{attribute 'reflection'} 
FUNCTION_BLOCK PUBLIC FB_Testsuites EXTENDS FB_Base IMPLEMENTS I_Testsuites
VAR_INPUT
	fbList:				FB_ListTestsuite;
END_VAR
VAR_OUTPUT
END_VAR
VAR
	stTestsuites:    	ST_Testsuites;
	bSave: 				BOOL;
	sFilePathName:		STRING(255):= 'C:\report.xml';

	fbXml:				FB_XmlDomParser;
	testsuites:			PVOID;
END_VAR

SUPER^();


fbXml.SaveDocumentToFile(sFilePathName, bSave);

METHOD PROTECTED M_Started : BOOL
VAR_INPUT
END_VAR

VAR
	nIndex: DINT;
END_VAR
M_Started:= TRUE;
WHILE nIndex < fbList.P_Length DO
	M_Started:= M_Started AND (fbList.M_Get(nIndex).P_State = E_Base.Stopped);
	nIndex:= nIndex + 1;
END_WHILE
END_METHOD

METHOD PROTECTED M_Starting : BOOL
VAR_INPUT
END_VAR

VAR
	nIndex: DINT;
END_VAR
CASE nState OF
	0:
		IF 	SUPER^.M_Starting() THEN
			fbXml.NewDocument();
			stTestsuites.sName:= M_GetName(sInstancePath);
			stTestsuites.nTests:= 0;
			stTestsuites.nFailures:= 0;
			stTestsuites.nErrors:= 0;
			stTestsuites.nSkipped:= 0;
			stTestsuites.nAssertions:= 0;
			stTestsuites.fTime:= 0.0;
			nState:= 1;
		END_IF
		
	1:
		testsuites:= fbXml.AppendNode(fbXml.GetDocumentNode(), 'testsuites');
		fbXml.AppendAttribute(testsuites, 'name', stTestsuites.sName);					// name        Name of the entire test run  
		fbXml.AppendAttributeAsInt(testsuites, 'tests', stTestsuites.nTests);			// tests       Total number of tests in this file    
		fbXml.AppendAttributeAsInt(testsuites, 'failures', stTestsuites.nFailures);		// failures    Total number of failed tests in this file 
		fbXml.AppendAttributeAsInt(testsuites, 'errors', stTestsuites.nErrors);			// errors      Total number of errored tests in this file     
		fbXml.AppendAttributeAsInt(testsuites, 'skipped', stTestsuites.nSkipped);		// skipped     Total number of skipped tests in this file    
		fbXml.AppendAttributeAsInt(testsuites, 'assertions', stTestsuites.nAssertions);	// assertions  Total number of assertions for all tests in this file    
		fbXml.AppendAttributeAsDouble(testsuites, 'time', stTestsuites.fTime);			// time        Aggregated time of all tests in this file in seconds     
		fbXml.AppendAttribute(testsuites, 'timestamp', stTestsuites.sTimestamp);			// timestamp   Date and time of when the test run was executed (in ISO 8601
		nState:= 2;
	
	2:
		WHILE nIndex < fbList.P_Length DO
			fbList.M_Get(nIndex).M_Request(E_Base.Starting);
			nIndex:= nIndex + 1;
		END_WHILE
		nState:= 3;
		
	3:
		M_Starting:= TRUE;
		
END_CASE
END_METHOD

METHOD PROTECTED M_Stopping : BOOL
VAR_INPUT
END_VAR
VAR
	nIndex: DINT;
	stTestsuite: ST_Testsuite;
END_VAR
CASE nState OF
	0:
		WHILE nIndex < fbList.P_Length DO
			stTestsuite:= fbList.M_Get(nIndex).P_Result;
			stTestsuites.nTests:= stTestsuites.nTests + stTestsuite.nTests;
			stTestsuites.nFailures:= stTestsuites.nFailures + stTestsuite.nFailures;
			stTestsuites.nErrors:= stTestsuites.nErrors + stTestsuite.nErrors;
			stTestsuites.nSkipped:= stTestsuites.nSkipped + stTestsuite.nSkipped;
			stTestsuites.nAssertions:= stTestsuites.nAssertions + stTestsuite.nAssertions;
			stTestsuites.fTime:= stTestsuites.fTime +  stTestsuite.fTime;
			fbXml.AppendCopy(testsuites, fbList.M_Get(nIndex).P_Node);
			nIndex:= nIndex + 1;
		END_WHILE
		nState:= 1;
		
	1:
		fbXml.SetAttribute(fbXml.Attribute(testsuites, 'name'), stTestsuites.sName);					
		fbXml.SetAttributeAsInt(fbXml.Attribute(testsuites, 'tests'), stTestsuites.nTests);			
		fbXml.SetAttributeAsInt(fbXml.Attribute(testsuites, 'failures'), stTestsuites.nFailures);		
		fbXml.SetAttributeAsInt(fbXml.Attribute(testsuites, 'errors'), stTestsuites.nErrors);			
		fbXml.SetAttributeAsInt(fbXml.Attribute(testsuites, 'skipped'), stTestsuites.nSkipped);		
		fbXml.SetAttributeAsInt(fbXml.Attribute(testsuites, 'assertions'), stTestsuites.nAssertions);	
		fbXml.SetAttributeAsDouble(fbXml.Attribute(testsuites, 'time'), stTestsuites.fTime);			
		fbXml.SetAttribute(fbXml.Attribute(testsuites, 'timestamp'), stTestsuites.sTimestamp);
		nState:= 2;
	
	2:
		bSave:= TRUE;
		nState:= 3;
		
	3:
		IF NOT bSave THEN
			nState:= 4;
		END_IF

	4:
		M_Stopping:= TRUE;
		
END_CASE
END_METHOD

END_FUNCTION_BLOCK

(* stored: Version 1.1.0.1
   POU FB_Testsuites: Id {f57812b9-99c8-4f64-b54a-807a33ca5cc6}, SpecialFunc None
   Method M_Started: Id {9f9f5ca1-441c-0f29-0c6d-16c04b2958a4}
   Method M_Starting: Id {a8b1fe70-9112-024f-0be9-355ea21512f0}
   Method M_Stopping: Id {188bbc9a-c2f6-0b60-00aa-0b55afe47559} *)
